FUNCTION_BLOCK PUBLIC FB_Foo
VAR_INPUT
END_VAR
VAR_OUTPUT
	{attribute 'init_namespace'}
	sNamespace	:	STRING;	
END_VAR
VAR
END_VAR

END_FUNCTION_BLOCK

(* stored: Version 1.1.0.1, ProductVersion 3.1.4020.6
   POU FB_Foo: Id {487d9a70-20eb-4815-a5f4-32a65a24001c}, SpecialFunc None *)
